# EPICS StreamDevice protocol: siteApps-725b29e158e8061764313f5708af9e46fe30c0a8/siteApps-725b29e158e8061764313f5708af9e46fe30c0a8/keithley6514/keithley6514Sup/devkeithley6514.proto
Terminator = CR LF;

getIDN
{
    out "*IDN?";
    in  "%\$1[^\r\n]";
    ExtraInput = Ignore;
}

cmd
{
    out "\$1";
}

getF
{
    out "\$1?";
    in  "%f";
    ExtraInput = Ignore;
}

setF
{
    out "\$1 %f";
#    @init { out "\$1?"; in "%f"; }
    @init { getF; }
}

getD
{
    out "\$1?";
    in  "%d";
    ExtraInput = Ignore;
}

setD
{
    out "\$1 %d";
#    @init { out "\$1?"; in "%d"; }
    @init { getD; }
}

setLocRem {
    out "SYST:%{LOC|REM}";
}

# CURR:RANGE?
# +2.100000E-04

getCurrentRange
{
    out "CURR:RANG?";
    in  "%*[^E]E-%d";
    ExtraInput = Ignore;
}

setCurrentRange
{
    out "CURR:RANG 2E-%d";
#    @init { out "CURR:RANG?"; in "%*[^E]E-%d"; }
    @init { getCurrentRange; }
}

# stringin
getFunc
{
    out "FUNC?";
    in  "%s";
    ExtraInput = Ignore;
}

# stringout
setFunc
{
    out "FUNC \'%s\'";
}

# stringin
getError
{
    out "SYST:ERR?";
    in  "%\$1[^\r\n]";
    ExtraInput = Ignore;
}

measureCurrent
{
    ReplyTimeout = 5000;
    out "READ?";
    in  "%f";
    ExtraInput = Ignore;
}

getLineF
{
    out "SYST:LFR?";
    in  "%d";
}

setLineF
{
    out "SYST:LFR %d";
#    @init { out "CURR:RANG?"; in "%*[^E]E-%d"; }
    @init { getLineF; }
}

##
##
##

setADRate
{
    out "CURR:NPLC %{6.00|1.00|0.10}";
    @init { out "CURR:NPLC?"; in "%{6.00|1.00|0.10}"; }
}

getADRate
{
    out "CURR:NPLC?";
    in  "%{6.00|1.00|0.10}";
    ExtraInput = Ignore;
}
